// TIA Portal V18 export
TYPE "FIODia"
// stored: IsFailsafeCompliant true
   STRUCT
      ModulePassOut : Bool;   // 模块钝化
      ModuleACK_REQ : Bool;   // 模块需确认重新集成
      Channel0PassOut : Bool;   // 通道0钝化
      Channel1PassOut : Bool;   // 通道1钝化
      Channel2PassOut : Bool;   // 通道2钝化
      Channel3PassOut : Bool;   // 通道3钝化
      Channel4PassOut : Bool;   // 通道4钝化
      Channel5PassOut : Bool;   // 通道5钝化
      Channel6PassOut : Bool;   // 通道6钝化
      Channel7PassOut : Bool;   // 通道7钝化
   END_STRUCT;
END_TYPE
